TYPE ST_ResD7 :
STRUCT
	PathID			:UINT;
	PathPresent		:BYTE;
	MotorIndex		:BYTE;
	MotorPresent	:BYTE;
	MotorType		:BYTE;
	MotorFaultData	:ARRAY[0..14] OF BYTE;
	CRC1			:BYTE;	    (* 1 byte*)
	CRC2			:BYTE;	    (* 1 byte*)
END_STRUCT
END_TYPE

(* stored: Version 1.1.0.1, ProductVersion 3.1.4020.12
   DUT ST_ResD7: Id {724622f8-e423-4d86-8cca-0c2d135e8ef2} *)
